// TwinCAT 3 PLC project SPS
// ProgramVersion: 3.1.4023.0
// libraries:
//   Tc2_Standard, * (Beckhoff Automation GmbH)
//   Tc2_System, * (Beckhoff Automation GmbH)
//   Tc2_TcpIp, * (Beckhoff Automation GmbH)
//   Tc2_Utilities, * (Beckhoff Automation GmbH)
//   Tc3_Module, * (Beckhoff Automation GmbH)
// project tree:
//   DUTs/ OBIS_Datatype.TcDUT
//   / PlcTask.TcTTO
//   POUs/ EL3443_OBIS.TcPOU, FB_OBIS.TcPOU, FB_SPEEDWIRE.TcPOU, MAIN.TcPOU, UnixTimestamp.TcPOU
// real-time tasks:
//   TASK PlcTask: cycle T#10ms, priority 20, ADS port 350
// I/O:
//   DEVICE Gerät 1 (EtherCAT), AmsNetId 172.17.204.224.2.1
//     Klemme 1 (EK1100) [EK1100 EtherCAT-Koppler (2A E-Bus)]
//       Klemme 2 (EL3443) [EL3443 3K. Leistungsmessung]
// variable links:
//   SPS/SPS Instance <-> Device 1 (EtherCAT)/Term 1 (EK1100)/Term 2 (EL3443)
//     PlcTask Inputs/MAIN.EL3443_Terminal.MDP5001_341_Input/MDP5001_341_L1_Basic_Current <-> L1 Basic/Current
//     PlcTask Inputs/MAIN.EL3443_Terminal.MDP5001_341_Input/MDP5001_341_L2_Basic_Current <-> L2 Basic/Current
//     PlcTask Inputs/MAIN.EL3443_Terminal.MDP5001_341_Input/MDP5001_341_L3_Basic_Current <-> L3 Basic/Current
//     PlcTask Inputs/MAIN.EL3443_Terminal.MDP5001_341_Input/MDP5001_341_L1_Basic_Voltage <-> L1 Basic/Voltage
//     PlcTask Inputs/MAIN.EL3443_Terminal.MDP5001_341_Input/MDP5001_341_L2_Basic_Voltage <-> L2 Basic/Voltage
//     PlcTask Inputs/MAIN.EL3443_Terminal.MDP5001_341_Input/MDP5001_341_L3_Basic_Voltage <-> L3 Basic/Voltage
//     PlcTask Inputs/MAIN.EL3443_Terminal.MDP5001_341_Input/MDP5001_341_L1_Power_Active_Power <-> L1 Power/Active Power
//     PlcTask Inputs/MAIN.EL3443_Terminal.MDP5001_341_Input/MDP5001_341_L2_Power_Active_Power <-> L2 Power/Active Power
//     PlcTask Inputs/MAIN.EL3443_Terminal.MDP5001_341_Input/MDP5001_341_L3_Power_Active_Power <-> L3 Power/Active Power
//     PlcTask Inputs/MAIN.EL3443_Terminal.MDP5001_341_Input/MDP5001_341_L1_Power_Apparent_Power <-> L1 Power/Apparent Power
//     PlcTask Inputs/MAIN.EL3443_Terminal.MDP5001_341_Input/MDP5001_341_L2_Power_Apparent_Power <-> L2 Power/Apparent Power
//     PlcTask Inputs/MAIN.EL3443_Terminal.MDP5001_341_Input/MDP5001_341_L3_Power_Apparent_Power <-> L3 Power/Apparent Power
//     PlcTask Inputs/MAIN.EL3443_Terminal.MDP5001_341_Input/MDP5001_341_L1_Power_Power_Factor <-> L1 Power/Power Factor
//     PlcTask Inputs/MAIN.EL3443_Terminal.MDP5001_341_Input/MDP5001_341_L2_Power_Power_Factor <-> L2 Power/Power Factor
//     PlcTask Inputs/MAIN.EL3443_Terminal.MDP5001_341_Input/MDP5001_341_L3_Power_Power_Factor <-> L3 Power/Power Factor
//     PlcTask Inputs/MAIN.EL3443_Terminal.MDP5001_341_Input/MDP5001_341_L1_Power_Reactive_Power <-> L1 Power/Reactive Power
//     PlcTask Inputs/MAIN.EL3443_Terminal.MDP5001_341_Input/MDP5001_341_L2_Power_Reactive_Power <-> L2 Power/Reactive Power
//     PlcTask Inputs/MAIN.EL3443_Terminal.MDP5001_341_Input/MDP5001_341_L3_Power_Reactive_Power <-> L3 Power/Reactive Power
//     PlcTask Inputs/MAIN.EL3443_Terminal.MDP5001_341_Input/MDP5001_341_L1_Status_Current_Guard_Error <-> L1 Status/Current Guard Error
//     PlcTask Inputs/MAIN.EL3443_Terminal.MDP5001_341_Input/MDP5001_341_L2_Status_Current_Guard_Error <-> L2 Status/Current Guard Error
//     PlcTask Inputs/MAIN.EL3443_Terminal.MDP5001_341_Input/MDP5001_341_L3_Status_Current_Guard_Error <-> L3 Status/Current Guard Error
//     PlcTask Inputs/MAIN.EL3443_Terminal.MDP5001_341_Input/MDP5001_341_L1_Status_Current_Guard_Warning <-> L1 Status/Current Guard Warning
//     PlcTask Inputs/MAIN.EL3443_Terminal.MDP5001_341_Input/MDP5001_341_L2_Status_Current_Guard_Warning <-> L2 Status/Current Guard Warning
//     PlcTask Inputs/MAIN.EL3443_Terminal.MDP5001_341_Input/MDP5001_341_L3_Status_Current_Guard_Warning <-> L3 Status/Current Guard Warning
//     PlcTask Inputs/MAIN.EL3443_Terminal.MDP5001_341_Input/MDP5001_341_L1_Status_Inaccurate_Current <-> L1 Status/Inaccurate Current
//     PlcTask Inputs/MAIN.EL3443_Terminal.MDP5001_341_Input/MDP5001_341_L2_Status_Inaccurate_Current <-> L2 Status/Inaccurate Current
//     PlcTask Inputs/MAIN.EL3443_Terminal.MDP5001_341_Input/MDP5001_341_L3_Status_Inaccurate_Current <-> L3 Status/Inaccurate Current
//     PlcTask Inputs/MAIN.EL3443_Terminal.MDP5001_341_Input/MDP5001_341_L1_Status_Inaccurate_Voltage <-> L1 Status/Inaccurate Voltage
//     PlcTask Inputs/MAIN.EL3443_Terminal.MDP5001_341_Input/MDP5001_341_L2_Status_Inaccurate_Voltage <-> L2 Status/Inaccurate Voltage
//     PlcTask Inputs/MAIN.EL3443_Terminal.MDP5001_341_Input/MDP5001_341_L3_Status_Inaccurate_Voltage <-> L3 Status/Inaccurate Voltage
//     PlcTask Inputs/MAIN.EL3443_Terminal.MDP5001_341_Input/MDP5001_341_L1_Status_Overcurrent <-> L1 Status/Overcurrent
//     PlcTask Inputs/MAIN.EL3443_Terminal.MDP5001_341_Input/MDP5001_341_L2_Status_Overcurrent <-> L2 Status/Overcurrent
//     PlcTask Inputs/MAIN.EL3443_Terminal.MDP5001_341_Input/MDP5001_341_L3_Status_Overcurrent <-> L3 Status/Overcurrent
//     PlcTask Inputs/MAIN.EL3443_Terminal.MDP5001_341_Input/MDP5001_341_L1_Status_Overvoltage <-> L1 Status/Overvoltage
//     PlcTask Inputs/MAIN.EL3443_Terminal.MDP5001_341_Input/MDP5001_341_L2_Status_Overvoltage <-> L2 Status/Overvoltage
//     PlcTask Inputs/MAIN.EL3443_Terminal.MDP5001_341_Input/MDP5001_341_L3_Status_Overvoltage <-> L3 Status/Overvoltage
//     PlcTask Inputs/MAIN.EL3443_Terminal.MDP5001_341_Input/MDP5001_341_L1_Status_TxPDO_Toggle <-> L1 Status/TxPDO Toggle
//     PlcTask Inputs/MAIN.EL3443_Terminal.MDP5001_341_Input/MDP5001_341_L2_Status_TxPDO_Toggle <-> L2 Status/TxPDO Toggle
//     PlcTask Inputs/MAIN.EL3443_Terminal.MDP5001_341_Input/MDP5001_341_L3_Status_TxPDO_Toggle <-> L3 Status/TxPDO Toggle
//     PlcTask Inputs/MAIN.EL3443_Terminal.MDP5001_341_Input/MDP5001_341_L1_Status_Voltage_Guard_Error <-> L1 Status/Voltage Guard Error
//     PlcTask Inputs/MAIN.EL3443_Terminal.MDP5001_341_Input/MDP5001_341_L2_Status_Voltage_Guard_Error <-> L2 Status/Voltage Guard Error
//     PlcTask Inputs/MAIN.EL3443_Terminal.MDP5001_341_Input/MDP5001_341_L3_Status_Voltage_Guard_Error <-> L3 Status/Voltage Guard Error
//     PlcTask Inputs/MAIN.EL3443_Terminal.MDP5001_341_Input/MDP5001_341_L1_Status_Voltage_Guard_Warning <-> L1 Status/Voltage Guard Warning
//     PlcTask Inputs/MAIN.EL3443_Terminal.MDP5001_341_Input/MDP5001_341_L2_Status_Voltage_Guard_Warning <-> L2 Status/Voltage Guard Warning
//     PlcTask Inputs/MAIN.EL3443_Terminal.MDP5001_341_Input/MDP5001_341_L3_Status_Voltage_Guard_Warning <-> L3 Status/Voltage Guard Warning
//     PlcTask Inputs/MAIN.EL3443_Terminal.MDP5001_341_Input/MDP5001_341_L1_Status_Voltage_Sign_Bit <-> L1 Status/Voltage Sign Bit
//     PlcTask Inputs/MAIN.EL3443_Terminal.MDP5001_341_Input/MDP5001_341_L2_Status_Voltage_Sign_Bit <-> L2 Status/Voltage Sign Bit
//     PlcTask Inputs/MAIN.EL3443_Terminal.MDP5001_341_Input/MDP5001_341_L3_Status_Voltage_Sign_Bit <-> L3 Status/Voltage Sign Bit
//     PlcTask Inputs/MAIN.EL3443_Terminal.MDP5001_341_Input/MDP5001_341_L3_Statistic_Current_Current_Peak <-> L3 Statistic Current/Current Peak
//     PlcTask Inputs/MAIN.EL3443_Terminal.MDP5001_341_Input/MDP5001_341_L3_Statistic_Current_Current_RMS_Maximum <-> L3 Statistic Current/Current RMS Maximum
//     PlcTask Inputs/MAIN.EL3443_Terminal.MDP5001_341_Input/MDP5001_341_L3_Statistic_Current_Current_RMS_Minimum <-> L3 Statistic Current/Current RMS Minimum
//     PlcTask Inputs/MAIN.EL3443_Terminal.MDP5001_341_Input/MDP5001_341_L3_Statistic_Power_Active_Power_Avg <-> L3 Statistic Power/Active Power Avg
//     PlcTask Inputs/MAIN.EL3443_Terminal.MDP5001_341_Input/MDP5001_341_L3_Statistic_Power_Active_Power_Max <-> L3 Statistic Power/Active Power Max
//     PlcTask Inputs/MAIN.EL3443_Terminal.MDP5001_341_Input/MDP5001_341_L3_Statistic_Power_Active_Power_Min <-> L3 Statistic Power/Active Power Min
//     PlcTask Inputs/MAIN.EL3443_Terminal.MDP5001_341_Input/MDP5001_341_L3_Statistic_Power_Apparent_Power_Avg <-> L3 Statistic Power/Apparent Power Avg
//     PlcTask Inputs/MAIN.EL3443_Terminal.MDP5001_341_Input/MDP5001_341_L3_Statistic_Power_Apparent_Power_Max <-> L3 Statistic Power/Apparent Power Max
//     PlcTask Inputs/MAIN.EL3443_Terminal.MDP5001_341_Input/MDP5001_341_L3_Statistic_Power_Apparent_Power_Min <-> L3 Statistic Power/Apparent Power Min
//     PlcTask Inputs/MAIN.EL3443_Terminal.MDP5001_341_Input/MDP5001_341_L3_Statistic_Power_Reactive_Power_Avg <-> L3 Statistic Power/Reactive Power Avg
//     PlcTask Inputs/MAIN.EL3443_Terminal.MDP5001_341_Input/MDP5001_341_L3_Statistic_Power_Reactive_Power_Max <-> L3 Statistic Power/Reactive Power Max
//     PlcTask Inputs/MAIN.EL3443_Terminal.MDP5001_341_Input/MDP5001_341_L3_Statistic_Power_Reactive_Power_Min <-> L3 Statistic Power/Reactive Power Min
//     PlcTask Inputs/MAIN.EL3443_Terminal.MDP5001_341_Input/MDP5001_341_Total_Active_Active_Energy <-> Total Active/Active Energy
//     PlcTask Inputs/MAIN.EL3443_Terminal.MDP5001_341_Input/MDP5001_341_Total_Active_Active_Negative_Energy <-> Total Active/Active Negative Energy
//     PlcTask Inputs/MAIN.EL3443_Terminal.MDP5001_341_Input/MDP5001_341_Total_Active_Active_Positive_Energy <-> Total Active/Active Positive Energy
//     PlcTask Inputs/MAIN.EL3443_Terminal.MDP5001_341_Input/MDP5001_341_Total_Active_Active_Power <-> Total Active/Active Power
//     PlcTask Inputs/MAIN.EL3443_Terminal.MDP5001_341_Input/MDP5001_341_Total_Apparent_Apparent_Energy <-> Total Apparent/Apparent Energy
//     PlcTask Inputs/MAIN.EL3443_Terminal.MDP5001_341_Input/MDP5001_341_Total_Apparent_Apparent_Negative_Energy <-> Total Apparent/Apparent Negative Energy
//     PlcTask Inputs/MAIN.EL3443_Terminal.MDP5001_341_Input/MDP5001_341_Total_Apparent_Apparent_Positive_Energy <-> Total Apparent/Apparent Positive Energy
//     PlcTask Inputs/MAIN.EL3443_Terminal.MDP5001_341_Input/MDP5001_341_Total_Apparent_Apparent_Power <-> Total Apparent/Apparent Power
//     PlcTask Inputs/MAIN.EL3443_Terminal.MDP5001_341_Input/MDP5001_341_Total_Basic_Calculated_Neutral_Line_Current <-> Total Basic/Calculated Neutral Line Current
//     PlcTask Inputs/MAIN.EL3443_Terminal.MDP5001_341_Input/MDP5001_341_Total_Basic_Frequency <-> Total Basic/Frequency
//     PlcTask Inputs/MAIN.EL3443_Terminal.MDP5001_341_Input/MDP5001_341_Total_Basic_Power_Factor <-> Total Basic/Power Factor
//     PlcTask Inputs/MAIN.EL3443_Terminal.MDP5001_341_Input/MDP5001_341_Total_Reactive_Reactive_Energy <-> Total Reactive/Reactive Energy
//     PlcTask Inputs/MAIN.EL3443_Terminal.MDP5001_341_Input/MDP5001_341_Total_Reactive_Reactive_Negative_Energy <-> Total Reactive/Reactive Negative Energy
//     PlcTask Inputs/MAIN.EL3443_Terminal.MDP5001_341_Input/MDP5001_341_Total_Reactive_Reactive_Positive_Energy <-> Total Reactive/Reactive Positive Energy
//     PlcTask Inputs/MAIN.EL3443_Terminal.MDP5001_341_Input/MDP5001_341_Total_Reactive_Reactive_Power <-> Total Reactive/Reactive Power
//     PlcTask Inputs/MAIN.EL3443_Terminal.MDP5001_341_Input/MDP5001_341_Total_Status_Active_Power_Guard_Error <-> Total Status/Active Power Guard Error
//     PlcTask Inputs/MAIN.EL3443_Terminal.MDP5001_341_Input/MDP5001_341_Total_Status_Active_Power_Guard_Warning <-> Total Status/Active Power Guard Warning
//     PlcTask Inputs/MAIN.EL3443_Terminal.MDP5001_341_Input/MDP5001_341_Total_Status_Apparent_Power_Guard_Error <-> Total Status/Apparent Power Guard Error
//     PlcTask Inputs/MAIN.EL3443_Terminal.MDP5001_341_Input/MDP5001_341_Total_Status_Apparent_Power_Guard_Warning <-> Total Status/Apparent Power Guard Warning
//     PlcTask Inputs/MAIN.EL3443_Terminal.MDP5001_341_Input/MDP5001_341_Total_Status_Frequency_Guard_Error <-> Total Status/Frequency Guard Error
//     PlcTask Inputs/MAIN.EL3443_Terminal.MDP5001_341_Input/MDP5001_341_Total_Status_Frequency_Guard_Warning <-> Total Status/Frequency Guard Warning
//     PlcTask Inputs/MAIN.EL3443_Terminal.MDP5001_341_Input/MDP5001_341_Total_Status_Grid_Direction <-> Total Status/Grid Direction
//     PlcTask Inputs/MAIN.EL3443_Terminal.MDP5001_341_Input/MDP5001_341_Total_Status_Neutral_Current_Guard_Error <-> Total Status/Neutral Current Guard Error
//     PlcTask Inputs/MAIN.EL3443_Terminal.MDP5001_341_Input/MDP5001_341_Total_Status_Neutral_Current_Guard_Warning <-> Total Status/Neutral Current Guard Warning
//     PlcTask Inputs/MAIN.EL3443_Terminal.MDP5001_341_Input/MDP5001_341_Total_Status_Power_Quality_Factor <-> Total Status/Power Quality Factor
//     PlcTask Inputs/MAIN.EL3443_Terminal.MDP5001_341_Input/MDP5001_341_Total_Status_Power_Quality_Guard_Error <-> Total Status/Power Quality Guard Error
//     PlcTask Inputs/MAIN.EL3443_Terminal.MDP5001_341_Input/MDP5001_341_Total_Status_Power_Quality_Guard_Warning <-> Total Status/Power Quality Guard Warning
//     PlcTask Inputs/MAIN.EL3443_Terminal.MDP5001_341_Input/MDP5001_341_Total_Status_System_State <-> Total Status/System State
//     PlcTask Inputs/MAIN.EL3443_Terminal.MDP5001_341_Input/MDP5001_341_Total_Status_TxPDO_State <-> Total Status/TxPDO State
//     PlcTask Inputs/MAIN.EL3443_Terminal.MDP5001_341_Input/MDP5001_341_Total_Status_TxPDO_Toggle <-> Total Status/TxPDO Toggle

CONFIGURATION SPS
    RESOURCE PLC ON TwinCAT3
        TASK PlcTask(INTERVAL := T#10ms, PRIORITY := 20);
        PROGRAM MAIN WITH PlcTask : MAIN;
    END_RESOURCE
END_CONFIGURATION

// ---- DUTs/OBIS_Datatype.TcDUT
{attribute 'qualified_only'}
{attribute 'strict'}
TYPE OBIS_Datatype :
(
	TOTAL_ActivePowerPositive := 0,
	TOTAL_ActivePowerNegative := 1,
	TOTAL_ActiveEnergyPositive := 2, 
	TOTAL_ActiveEnergyNegative := 3,
	TOTAL_ApparentPowerPositive := 4,
	TOTAL_ApparentPowerNegative := 5,
	TOTAL_ApparentEnergyPositive := 6, 
	TOTAL_ApparentEnergyNegative := 7,
	TOTAL_ReactivePowerPositive := 8,
	TOTAL_ReactivePowerNegative := 9,
	TOTAL_ReactiveEnergyPositive := 10, 
	TOTAL_ReactiveEnergyNegative := 11,
	TOTAL_PowerFactor := 12,
	TOTAL_Frequency := 13, 
	
	L1_ActivePowerPositive := 14,
	L1_ActivePowerNegative := 15,
	L1_ActiveEnergyPositive := 16, 
	L1_ActiveEnergyNegative := 17,
	L1_ApparentPowerPositive := 18,
	L1_ApparentPowerNegative := 19,
	L1_ApparentEnergyPositive := 20, 
	L1_ApparentEnergyNegative := 21,
	L1_ReactivePowerPositive := 22,
	L1_ReactivePowerNegative := 23,
	L1_ReactiveEnergyPositive := 24, 
	L1_ReactiveEnergyNegative := 25,
	L1_Current := 26,
	L1_Voltage := 27,
	L1_PowerFactor := 28,
	
	L2_ActivePowerPositive := 29,
	L2_ActivePowerNegative := 30,
	L2_ActiveEnergyPositive := 31, 
	L2_ActiveEnergyNegative := 32,
	L2_ApparentPowerPositive := 33,
	L2_ApparentPowerNegative := 34,
	L2_ApparentEnergyPositive := 35, 
	L2_ApparentEnergyNegative := 36,
	L2_ReactivePowerPositive := 37,
	L2_ReactivePowerNegative := 38,
	L2_ReactiveEnergyPositive := 39, 
	L2_ReactiveEnergyNegative := 40,
	L2_Current := 41,
	L2_Voltage := 42,
	L2_PowerFactor := 43,
	
	L3_ActivePowerPositive := 44,
	L3_ActivePowerNegative := 45,
	L3_ActiveEnergyPositive := 46, 
	L3_ActiveEnergyNegative := 47,
	L3_ApparentPowerPositive := 48,
	L3_ApparentPowerNegative := 49,
	L3_ApparentEnergyPositive := 50, 
	L3_ApparentEnergyNegative := 51,
	L3_ReactivePowerPositive := 52,
	L3_ReactivePowerNegative := 53,
	L3_ReactiveEnergyPositive := 54, 
	L3_ReactiveEnergyNegative := 55,
	L3_Current := 56,
	L3_Voltage := 57,
	L3_PowerFactor := 58
	
	
);
END_TYPE

// ---- POUs/MAIN.TcPOU
PROGRAM MAIN
VAR
	//Devices
	EL3443_Terminal			: MDP5001_341_A3044239;
	fbspeedwire				: FB_SPEEDWIRE;
END_VAR

fbspeedwire(
	EL3443 := EL3443_Terminal
	);

END_PROGRAM

// ---- POUs/FB_SPEEDWIRE.TcPOU
FUNCTION_BLOCK FB_SPEEDWIRE
VAR_INPUT
	bEnable					: BOOL 	:= TRUE;
	nLocalPort				: UDINT := 9522;
	sLocalHost				: T_IPv4Addr := '192.168.0.227';(* Adapt local IP address to your device *)
	nRemotePort				: UDINT := 9522;
	sMulticastAddr			: T_IPv4Addr := '239.12.255.254';
	
	EL3443		: MDP5001_341_A3044239;
END_VAR
VAR_OUTPUT
END_VAR
VAR
	fbUdpCreate 			: FB_SocketUdpCreate;
	fbSocketAddMulticast 	: FB_SocketUdpAddMulticastAddress;
	fbSocketDropMulticast 	: FB_SocketUdpDropMulticastAddress;
	fbSocketSend  			: FB_SocketUdpSendTo;
	fbSocketReceive 		: FB_SocketUdpReceiveFrom;
	fbSocketClose			: FB_SocketClose;
	fbCloseAll				: FB_SocketCloseAll;
	bInitialize				: BOOL := TRUE;
	bUdpCreated				: BOOL;
	bMulticastAdded			: BOOL; 
	
	nCounterIn 				: UDINT;
	nCounterOut 			: UDINT;
	nState 					: INT;		
	
	fbEL3443_2_OBIS			: EL3443_OBIS;
	
	send_ton 				: TON;
END_VAR

IF bInitialize = TRUE THEN
(* On PLC reset or program download close all opened/created sockets *)
	fbCloseAll( bExecute:= bInitialize );
	IF fbCloseAll.bBusy OR fbCloseAll.bError THEN
	//	RETURN;
	END_IF
	bInitialize := FALSE;
END_IF






CASE nState OF
0:
	IF bEnable THEN
		bUdpCreated := FALSE;
		bMulticastAdded := FALSE;
		nState := 1;
	END_IF
1:
	fbUdpCreate( bExecute := FALSE );
	fbUdpCreate( nLocalPort := nLocalPort, sLocalHost := sLocalHost, bExecute := TRUE);
	nState := 2;
2:
	fbUdpCreate( bExecute := FALSE );
	IF NOT fbUdpCreate.bBusy THEN
		IF NOT fbUdpCreate.bError THEN
			bUdpCreated := TRUE;
			fbSocketAddMulticast( bExecute := FALSE );
			fbSocketAddMulticast( hSocket := fbUdpCreate.hSocket, sMulticastAddr := sMulticastAddr, bExecute := TRUE );
			nState := 3;
		ELSE
			nState := 100;
		END_IF
	END_IF
3:
	fbSocketAddMulticast( bExecute := FALSE );
	IF NOT fbSocketAddMulticast.bBusy THEN
		IF NOT fbSocketAddMulticast.bError THEN
			bMulticastAdded := TRUE;
			nState := 4;
		ELSE
			nState := 100;
		END_IF
	END_IF
	
4:
	IF bEnable THEN
		nCounterOut := nCounterOut + 1;
		fbSocketSend( bExecute := FALSE );
		fbEL3443_2_OBIS(EL3443 := EL3443);
		fbSocketSend( nRemotePort := nRemotePort, sRemoteHost := sMulticastAddr, hSocket := fbUdpCreate.hSocket, cbLen:= fbEL3443_2_OBIS.GetDataLength(), pSrc := fbEL3443_2_OBIS.GetData(), bExecute := TRUE );
		nState := 5;
	ELSE
		nState := 10;
	END_IF
5:
	fbSocketSend( bExecute := FALSE );
	IF NOT fbSocketSend.bBusy THEN
		IF NOT fbSocketSend.bError THEN
			nState := 6;
		ELSE
 			nState := 100;
		END_IF
	END_IF
6:	
	fbSocketReceive( bExecute := FALSE );
	IF NOT fbSocketReceive.bBusy THEN
		IF NOT fbSocketReceive.bError THEN
			nState:= 7;
			
		ELSE
			nState := 100;
		END_IF
	END_IF

7:	send_ton(IN := TRUE, PT:= T#200MS);
	IF send_ton.Q THEN
		nState:= 4;
		send_ton(IN:=FALSE);
	END_IF
	
10:
	fbSocketDropMulticast( bExecute := FALSE );
	fbSocketDropMulticast( hSocket := fbUdpCreate.hSocket, sMulticastAddr := sMulticastAddr, bExecute := TRUE );
	nState := 11;
11:	
	fbSocketDropMulticast( bExecute := FALSE );
	IF NOT fbSocketDropMulticast.bBusy THEN
		bMulticastAdded := FALSE;
		IF NOT fbSocketDropMulticast.bError THEN
			nState := 20;
		ELSE
			nState := 100;
		END_IF
	END_IF

20:	
	fbSocketClose( bExecute := FALSE );
	fbSocketClose( hSocket := fbUdpCreate.hSocket, bExecute := TRUE );
	nState := 21;
21:	
	fbSocketClose( bExecute := FALSE );
	IF NOT fbSocketClose.bBusy THEN
		bUdpCreated := FALSE;
		IF NOT fbSocketClose.bError THEN
			nState := 0;	
		ELSE
			nState := 100;	
		END_IF
	END_IF
	
100:
	IF bMulticastAdded THEN
		nState := 10;
	ELSIF bUdpCreated THEN
		nState := 20;
	ELSE
		nState := 0;
	END_IF
	
END_CASE

END_FUNCTION_BLOCK

// ---- POUs/EL3443_OBIS.TcPOU
FUNCTION_BLOCK EL3443_OBIS
VAR_INPUT
	EL3443 : MDP5001_341_A3044239;
END_VAR
VAR_OUTPUT
END_VAR
VAR
	unixTime: UnixTimestamp;
    timestampSeconds: ULINT;
    timestampMilliseconds: ULINT;
	
	obis_data : FB_OBIS;	
END_VAR

unixTime();
timestampMilliseconds := unixTime.milliseconds;
timestampSeconds := unixTime.seconds;

obis_data.addTime(u32time := ULINT_TO_UDINT(timestampMilliseconds));

//L1------------------------------------------------

obis_data.Addfloat(datatype := OBIS_Datatype.L1_Voltage, floatdata := EL3443.MDP5001_341_Input.MDP5001_341_L1_Basic_Voltage);
obis_data.Addfloat(datatype := OBIS_Datatype.L1_Current, floatdata := EL3443.MDP5001_341_Input.MDP5001_341_L1_Basic_Current);
obis_data.Addfloat(datatype := OBIS_Datatype.L1_PowerFactor, floatdata := EL3443.MDP5001_341_Input.MDP5001_341_L1_Power_Power_Factor);

IF EL3443.MDP5001_341_Input.MDP5001_341_L1_Power_Active_Power > 0.0 THEN
	obis_data.Addfloat(datatype := OBIS_Datatype.L1_ActivePowerPositive, floatdata := EL3443.MDP5001_341_Input.MDP5001_341_L1_Power_Active_Power);
	obis_data.Addfloat(datatype := OBIS_Datatype.L1_ActivePowerNegative, floatdata := 0.0);
ELSE
	obis_data.Addfloat(datatype := OBIS_Datatype.L1_ActivePowerPositive, floatdata := 0.0);
	obis_data.Addfloat(datatype := OBIS_Datatype.L1_ActivePowerNegative, floatdata := -EL3443.MDP5001_341_Input.MDP5001_341_L1_Power_Active_Power);	
END_IF

IF EL3443.MDP5001_341_Input.MDP5001_341_L1_Power_Apparent_Power > 0.0 THEN
	obis_data.Addfloat(datatype := OBIS_Datatype.L1_ApparentPowerPositive, floatdata := EL3443.MDP5001_341_Input.MDP5001_341_L1_Power_Apparent_Power);
	obis_data.Addfloat(datatype := OBIS_Datatype.L1_ApparentPowerNegative, floatdata := 0.0);
ELSE
	obis_data.Addfloat(datatype := OBIS_Datatype.L1_ApparentPowerPositive, floatdata := 0.0);
	obis_data.Addfloat(datatype := OBIS_Datatype.L1_ApparentPowerNegative, floatdata := -EL3443.MDP5001_341_Input.MDP5001_341_L1_Power_Apparent_Power);	
END_IF

IF EL3443.MDP5001_341_Input.MDP5001_341_L1_Power_Reactive_Power > 0.0 THEN
	obis_data.Addfloat(datatype := OBIS_Datatype.L1_ReactivePowerPositive, floatdata := EL3443.MDP5001_341_Input.MDP5001_341_L1_Power_Reactive_Power);
	obis_data.Addfloat(datatype := OBIS_Datatype.L1_ReactivePowerNegative, floatdata := 0.0);
ELSE
	obis_data.Addfloat(datatype := OBIS_Datatype.L1_ReactivePowerPositive, floatdata := 0.0);
	obis_data.Addfloat(datatype := OBIS_Datatype.L1_ReactivePowerNegative, floatdata := -EL3443.MDP5001_341_Input.MDP5001_341_L1_Power_Reactive_Power);	
END_IF


(*
obis_data.AddUint64(datatype := OBIS_Datatype.L1_ActiveEnergyPositive, u64data := 0);
obis_data.AddUint64(datatype := OBIS_Datatype.L1_ActiveEnergyNegative, u64data := 0);
obis_data.AddUint64(datatype := OBIS_Datatype.L1_ApparentEnergyPositive, u64data := 0);
obis_data.AddUint64(datatype := OBIS_Datatype.L1_ApparentEnergyNegative, u64data := 0);
obis_data.AddUint64(datatype := OBIS_Datatype.L1_ReactiveEnergyPositive, u64data := 0);
obis_data.AddUint64(datatype := OBIS_Datatype.L1_ReactiveEnergyNegative, u64data := 0);

*)

//L2------------------------------------------------

obis_data.Addfloat(datatype := OBIS_Datatype.L2_Voltage, floatdata := EL3443.MDP5001_341_Input.MDP5001_341_L2_Basic_Voltage);
obis_data.Addfloat(datatype := OBIS_Datatype.L2_Current, floatdata := EL3443.MDP5001_341_Input.MDP5001_341_L2_Basic_Current);
obis_data.Addfloat(datatype := OBIS_Datatype.L2_PowerFactor, floatdata := EL3443.MDP5001_341_Input.MDP5001_341_L2_Power_Power_Factor);

IF EL3443.MDP5001_341_Input.MDP5001_341_L2_Power_Active_Power > 0.0 THEN
	obis_data.Addfloat(datatype := OBIS_Datatype.L2_ActivePowerPositive, floatdata := EL3443.MDP5001_341_Input.MDP5001_341_L2_Power_Active_Power);
	obis_data.Addfloat(datatype := OBIS_Datatype.L2_ActivePowerNegative, floatdata := 0.0);
ELSE
	obis_data.Addfloat(datatype := OBIS_Datatype.L2_ActivePowerPositive, floatdata := 0.0);
	obis_data.Addfloat(datatype := OBIS_Datatype.L2_ActivePowerNegative, floatdata := -EL3443.MDP5001_341_Input.MDP5001_341_L2_Power_Active_Power);	
END_IF

IF EL3443.MDP5001_341_Input.MDP5001_341_L2_Power_Apparent_Power > 0.0 THEN
	obis_data.Addfloat(datatype := OBIS_Datatype.L2_ApparentPowerPositive, floatdata := EL3443.MDP5001_341_Input.MDP5001_341_L2_Power_Apparent_Power);
	obis_data.Addfloat(datatype := OBIS_Datatype.L2_ApparentPowerNegative, floatdata := 0.0);
ELSE
	obis_data.Addfloat(datatype := OBIS_Datatype.L2_ApparentPowerPositive, floatdata := 0.0);
	obis_data.Addfloat(datatype := OBIS_Datatype.L2_ApparentPowerNegative, floatdata := -EL3443.MDP5001_341_Input.MDP5001_341_L2_Power_Apparent_Power);	
END_IF

IF EL3443.MDP5001_341_Input.MDP5001_341_L2_Power_Reactive_Power > 0.0 THEN
	obis_data.Addfloat(datatype := OBIS_Datatype.L2_ReactivePowerPositive, floatdata := EL3443.MDP5001_341_Input.MDP5001_341_L2_Power_Reactive_Power);
	obis_data.Addfloat(datatype := OBIS_Datatype.L2_ReactivePowerNegative, floatdata := 0.0);
ELSE
	obis_data.Addfloat(datatype := OBIS_Datatype.L2_ReactivePowerPositive, floatdata := 0.0);
	obis_data.Addfloat(datatype := OBIS_Datatype.L2_ReactivePowerNegative, floatdata := -EL3443.MDP5001_341_Input.MDP5001_341_L2_Power_Reactive_Power);	
END_IF

(*
obis_data.AddUint64(datatype := OBIS_Datatype.L2_ActiveEnergyPositive, u64data := 0);
obis_data.AddUint64(datatype := OBIS_Datatype.L2_ActiveEnergyNegative, u64data := 0);
obis_data.AddUint64(datatype := OBIS_Datatype.L2_ApparentEnergyPositive, u64data := 0);
obis_data.AddUint64(datatype := OBIS_Datatype.L2_ApparentEnergyNegative, u64data := 0);
obis_data.AddUint64(datatype := OBIS_Datatype.L2_ReactiveEnergyPositive, u64data := 0);
obis_data.AddUint64(datatype := OBIS_Datatype.L2_ReactiveEnergyNegative, u64data := 0);
*)

//L3------------------------------------------------

obis_data.Addfloat(datatype := OBIS_Datatype.L3_Voltage, floatdata := EL3443.MDP5001_341_Input.MDP5001_341_L3_Basic_Voltage);
obis_data.Addfloat(datatype := OBIS_Datatype.L3_Current, floatdata := EL3443.MDP5001_341_Input.MDP5001_341_L3_Basic_Current);
obis_data.Addfloat(datatype := OBIS_Datatype.L3_PowerFactor, floatdata := EL3443.MDP5001_341_Input.MDP5001_341_L3_Power_Power_Factor);

IF EL3443.MDP5001_341_Input.MDP5001_341_L3_Power_Active_Power > 0.0 THEN
	obis_data.Addfloat(datatype := OBIS_Datatype.L3_ActivePowerPositive, floatdata := EL3443.MDP5001_341_Input.MDP5001_341_L3_Power_Active_Power);
	obis_data.Addfloat(datatype := OBIS_Datatype.L3_ActivePowerNegative, floatdata := 0.0);
ELSE
	obis_data.Addfloat(datatype := OBIS_Datatype.L3_ActivePowerPositive, floatdata := 0.0);
	obis_data.Addfloat(datatype := OBIS_Datatype.L3_ActivePowerNegative, floatdata := -EL3443.MDP5001_341_Input.MDP5001_341_L3_Power_Active_Power);	
END_IF

IF EL3443.MDP5001_341_Input.MDP5001_341_L3_Power_Apparent_Power > 0.0 THEN
	obis_data.Addfloat(datatype := OBIS_Datatype.L3_ApparentPowerPositive, floatdata := EL3443.MDP5001_341_Input.MDP5001_341_L3_Power_Apparent_Power);
	obis_data.Addfloat(datatype := OBIS_Datatype.L3_ApparentPowerNegative, floatdata := 0.0);
ELSE
	obis_data.Addfloat(datatype := OBIS_Datatype.L3_ApparentPowerPositive, floatdata := 0.0);
	obis_data.Addfloat(datatype := OBIS_Datatype.L3_ApparentPowerNegative, floatdata := -EL3443.MDP5001_341_Input.MDP5001_341_L3_Power_Apparent_Power);	
END_IF

IF EL3443.MDP5001_341_Input.MDP5001_341_L3_Power_Reactive_Power > 0.0 THEN
	obis_data.Addfloat(datatype := OBIS_Datatype.L3_ReactivePowerPositive, floatdata := EL3443.MDP5001_341_Input.MDP5001_341_L3_Power_Reactive_Power);
	obis_data.Addfloat(datatype := OBIS_Datatype.L3_ReactivePowerNegative, floatdata := 0.0);
ELSE
	obis_data.Addfloat(datatype := OBIS_Datatype.L3_ReactivePowerPositive, floatdata := 0.0);
	obis_data.Addfloat(datatype := OBIS_Datatype.L3_ReactivePowerNegative, floatdata := -EL3443.MDP5001_341_Input.MDP5001_341_L3_Power_Reactive_Power);	
END_IF

(*
obis_data.AddUint64(datatype := OBIS_Datatype.L3_ActiveEnergyPositive, u64data := 0);
obis_data.AddUint64(datatype := OBIS_Datatype.L3_ActiveEnergyNegative, u64data := 0);
obis_data.AddUint64(datatype := OBIS_Datatype.L3_ApparentEnergyPositive, u64data := 0);
obis_data.AddUint64(datatype := OBIS_Datatype.L3_ApparentEnergyNegative, u64data := 0);
obis_data.AddUint64(datatype := OBIS_Datatype.L3_ReactiveEnergyPositive, u64data := 0);
obis_data.AddUint64(datatype := OBIS_Datatype.L3_ReactiveEnergyNegative, u64data := 0);
*)

//Total------------------------------------------------


obis_data.Addfloat(datatype := OBIS_Datatype.TOTAL_PowerFactor, floatdata := EL3443.MDP5001_341_Input.MDP5001_341_Total_Basic_Power_Factor);
obis_data.Addfloat(datatype := OBIS_Datatype.TOTAL_Frequency, floatdata := EL3443.MDP5001_341_Input.MDP5001_341_Total_Basic_Frequency);

(*
obis_data.AddUint64(datatype := OBIS_Datatype.TOTAL_ActiveEnergyPositive, u64data := EL3443.MDP5001_341_Input.MDP5001_341_Total_Active_Active_Positive_Energy);
obis_data.AddUint64(datatype := OBIS_Datatype.TOTAL_ActiveEnergyNegative, u64data := EL3443.MDP5001_341_Input.MDP5001_341_Total_Active_Active_Negative_Energy);
obis_data.AddUint64(datatype := OBIS_Datatype.TOTAL_ApparentEnergyPositive, u64data := EL3443.MDP5001_341_Input.MDP5001_341_Total_Apparent_Apparent_Positive_Energy);
obis_data.AddUint64(datatype := OBIS_Datatype.TOTAL_ApparentEnergyNegative, u64data := EL3443.MDP5001_341_Input.MDP5001_341_Total_Apparent_Apparent_Negative_Energy);
obis_data.AddUint64(datatype := OBIS_Datatype.TOTAL_ReactiveEnergyPositive, u64data := EL3443.MDP5001_341_Input.MDP5001_341_Total_Reactive_Reactive_Positive_Energy);
obis_data.AddUint64(datatype := OBIS_Datatype.TOTAL_ReactiveEnergyNegative, u64data := EL3443.MDP5001_341_Input.MDP5001_341_Total_Reactive_Reactive_Negative_Energy);
*)

IF EL3443.MDP5001_341_Input.MDP5001_341_Total_Active_Active_Power > 0.0 THEN
	obis_data.Addfloat(datatype := OBIS_Datatype.TOTAL_ActivePowerPositive, floatdata := EL3443.MDP5001_341_Input.MDP5001_341_Total_Active_Active_Power);
	obis_data.Addfloat(datatype := OBIS_Datatype.TOTAL_ActivePowerNegative, floatdata := 0.0);
ELSE
	obis_data.Addfloat(datatype := OBIS_Datatype.TOTAL_ActivePowerPositive, floatdata := 0.0);
	obis_data.Addfloat(datatype := OBIS_Datatype.TOTAL_ActivePowerNegative, floatdata := -EL3443.MDP5001_341_Input.MDP5001_341_Total_Active_Active_Power);	
END_IF

IF EL3443.MDP5001_341_Input.MDP5001_341_Total_Apparent_Apparent_Power > 0.0 THEN
	obis_data.Addfloat(datatype := OBIS_Datatype.TOTAL_ApparentPowerPositive, floatdata := EL3443.MDP5001_341_Input.MDP5001_341_Total_Apparent_Apparent_Power);
	obis_data.Addfloat(datatype := OBIS_Datatype.TOTAL_ApparentPowerNegative, floatdata := 0.0);
ELSE
	obis_data.Addfloat(datatype := OBIS_Datatype.TOTAL_ApparentPowerPositive, floatdata := 0.0);
	obis_data.Addfloat(datatype := OBIS_Datatype.TOTAL_ApparentPowerNegative, floatdata := -EL3443.MDP5001_341_Input.MDP5001_341_Total_Apparent_Apparent_Power);	
END_IF

IF EL3443.MDP5001_341_Input.MDP5001_341_Total_Reactive_Reactive_Power > 0.0 THEN
	obis_data.Addfloat(datatype := OBIS_Datatype.TOTAL_ReactivePowerPositive, floatdata := EL3443.MDP5001_341_Input.MDP5001_341_Total_Reactive_Reactive_Power);
	obis_data.Addfloat(datatype := OBIS_Datatype.TOTAL_ReactivePowerNegative, floatdata := 0.0);
ELSE
	obis_data.Addfloat(datatype := OBIS_Datatype.TOTAL_ReactivePowerPositive, floatdata := 0.0);
	obis_data.Addfloat(datatype := OBIS_Datatype.TOTAL_ReactivePowerNegative, floatdata := -EL3443.MDP5001_341_Input.MDP5001_341_Total_Reactive_Reactive_Power);	
END_IF

METHOD GetData : POINTER TO BYTE
VAR_INPUT
END_VAR
GetData := obis_data.GetData();
END_METHOD

METHOD GetDataLength : UDINT
VAR_INPUT
END_VAR
GetDataLength := 608;
END_METHOD

END_FUNCTION_BLOCK

// ---- POUs/UnixTimestamp.TcPOU
FUNCTION_BLOCK UnixTimestamp
VAR_INPUT
END_VAR
VAR_OUTPUT
	seconds: ULINT;
    milliseconds: ULINT;
END_VAR
VAR
	localSystemTime : FB_LocalSystemTime := ( bEnable := TRUE, dwCycle := 1 );
    getTimeZoneInformation : FB_GetTimeZoneInformation;
    timeZoneInformation : ST_TimeZoneInformation;
    specificLocalTimeToFileTime : FB_TzSpecificLocalTimeToFileTime;
    fileTime: T_FILETIME;
    onZerothSecondLastCycle : BOOL;
END_VAR

// Get local system time
localSystemTime();

// On the zeroth second of each minutesync timezone information
IF (timeZoneInformation.standardName = '' OR (localSystemTime.systemTime.wSecond = 0 AND NOT onZerothSecondLastCycle)) THEN
    getTimeZoneInformation(sNetID := '', bExecute := TRUE, tzInfo => timeZoneInformation);
END_IF;

// Convert local system time to unix timestamps
specificLocalTimeToFileTime(in := Tc2_Utilities.SYSTEMTIME_TO_FILETIME(localSystemTime.systemTime), tzInfo := timeZoneInformation, out => fileTime);
seconds := (SHL(DWORD_TO_ULINT(fileTime.dwHighDateTime), 32) + DWORD_TO_ULINT(fileTime.dwLowDateTime)) / 10000000 - 11644473600;
milliseconds := (SHL(DWORD_TO_ULINT(fileTime.dwHighDateTime), 32) + DWORD_TO_ULINT(fileTime.dwLowDateTime)) / 10000 - 11644473600000;

onZerothSecondLastCycle := localSystemTime.systemTime.wSecond = 0;

END_FUNCTION_BLOCK

// ---- POUs/FB_OBIS.TcPOU
FUNCTION_BLOCK FB_OBIS
VAR_INPUT
END_VAR
VAR_OUTPUT
END_VAR
VAR
	data : ARRAY [0..607] OF BYTE := [83, 77, 65, 0, 0, 4, 2, 160, 0, 0, 0, 1, 2, 76, 0, 16, 96, 105, 1, 93, 113, 87, 157, 42, 145, 195, 170, 229, 0, 1, 4, 0, 0, 0, 4, 192, 0, 1, 8, 0, 0, 0, 0, 1, 27, 80, 113, 64, 0, 2, 4, 0, 0, 0, 0, 0, 0, 2, 8, 0, 0, 0, 0, 0, 65, 115, 204, 96, 0, 3, 4, 0, 0, 0, 0, 0, 0, 3, 8, 0, 0, 0, 0, 0, 1, 68, 24, 192, 0, 4, 4, 0, 0, 0, 7, 97, 0, 4, 8, 0, 0, 0, 0, 0, 203, 199, 123, 0, 0, 9, 4, 0, 0, 0, 8, 198, 0, 9, 8, 0, 0, 0, 0, 1, 121, 25, 106, 32, 0, 10, 4, 0, 0, 0, 0, 0, 0, 10, 8, 0, 0, 0, 0, 0, 70, 76, 180, 64, 0, 13, 4, 0, 0, 0, 2, 28, 0, 14, 4, 0, 0, 0, 195, 240, 0, 21, 4, 0, 0, 0, 0, 0, 0, 21, 8, 0, 0, 0, 0, 0, 72, 109, 19, 160, 0, 22, 4, 0, 0, 0, 0, 217, 0, 22, 8, 0, 0, 0, 0, 0, 30, 95, 6, 64, 0, 23, 4, 0, 0, 0, 0, 0, 0, 23, 8, 0, 0, 0, 0, 0, 0, 136, 59, 0, 0, 24, 4, 0, 0, 0, 0, 223, 0, 24, 8, 0, 0, 0, 0, 0, 37, 222, 86, 0, 0, 29, 4, 0, 0, 0, 0, 0, 0, 29, 8, 0, 0, 0, 0, 0, 101, 164, 5, 0, 0, 30, 4, 0, 0, 0, 1, 55, 0, 30, 8, 0, 0, 0, 0, 0, 30, 244, 112, 63, 0, 31, 4, 0, 0, 0, 0, 180, 0, 32, 4, 0, 0, 3, 138, 34, 0, 33, 4, 0, 0, 0, 2, 188, 0, 41, 4, 0, 0, 0, 6, 72, 0, 41, 8, 0, 0, 0, 0, 0, 166, 88, 167, 224, 0, 42, 4, 0, 0, 0, 0, 0, 0, 42, 8, 0, 0, 0, 0, 0, 16, 177, 174, 128, 0, 43, 4, 0, 0, 0, 0, 0, 0, 43, 8, 0, 0, 0, 0, 0, 1, 149, 101, 64, 0, 44, 4, 0, 0, 0, 4, 236, 0, 44, 8, 0, 0, 0, 0, 0, 114, 214, 221, 96, 0, 49, 4, 0, 0, 0, 7, 251, 0, 49, 8, 0, 0, 0, 0, 0, 209, 9, 218, 224, 0, 50, 4, 0, 0, 0, 0, 0, 0, 50, 8, 0, 0, 0, 0, 0, 19, 30, 104, 192, 0, 51, 4, 0, 0, 0, 4, 96, 0, 52, 4, 0, 0, 3, 133, 4, 0, 53, 4, 0, 0, 0, 3, 22, 0, 61, 4, 0, 0, 0, 0, 0, 0, 61, 8, 0, 0, 0, 0, 0, 58, 50, 2, 159, 0, 62, 4, 0, 0, 0, 0, 176, 0, 62, 8, 0, 0, 0, 0, 0, 32, 9, 215, 224, 0, 63, 4, 0, 0, 0, 0, 0, 0, 63, 8, 0, 0, 0, 0, 0, 0, 93, 98, 64, 0, 64, 4, 0, 0, 0, 1, 150, 0, 64, 8, 0, 0, 0, 0, 0, 52, 73, 49, 96, 0, 69, 4, 0, 0, 0, 0, 0, 0, 69, 8, 0, 0, 0, 0, 0, 93, 66, 99, 192, 0, 70, 4, 0, 0, 0, 1, 187, 0, 70, 8, 0, 0, 0, 0, 0, 33, 166, 237, 224, 0, 71, 4, 0, 0, 0, 0, 230, 0, 72, 4, 0, 0, 3, 130, 202, 0, 73, 4, 0, 0, 0, 1, 144, 144, 0, 0, 0, 2, 0, 18, 82, 0, 0, 0, 0];
	u32tmp : UDINT;
END_VAR


//sma signature
//data[0..3] = 83, 77, 65, 0, 

//sma tag0
//data[4..7] = 0, 4, 2, 160,

//sma group
//data[8..11] = 0, 0, 0, 1, 

//sma length offset
//data[12..13] =  2, 76,

//sma netver
//data[14..15] =  0, 16,

//sma protocol 
//data[16..17] = 96, 105

///Speedwire protocol
//SusyID
//data[18..19] = 1, 93

//SerialNumber
//data[20..23] = 113, 87, 157, 42, 

//Time
//data[24..27] = 145, 195, 170, 229,

//Total active power positive (8byte)
//data[28..35] = 0, 1, 4, 0, 0, 0, 4, 192,

//Total active enregy positive (12 byte)
//data[36..47] =  0, 1, 8, 0, 0, 0, 0, 1, 27, 80, 113, 64,

//Total active power negative (8byte)
//data[48..55] =  0, 2, 4, 0, 0, 0, 0, 0, 

//Total active enregy negative (12 byte)
//data[56..67] = 0,2, 8, 0, 0, 0, 0, 0, 65, 115, 204, 96,

//Total reactive power positive (8 byte)
// data[68..75] = 0, 3, 4, 0, 0, 0, 0, 0,

//Total reactive enegry pisitve (12 byte)
// data[76..87] = 0, 3, 8, 0, 0, 0, 0, 0, 1, 68, 24, 192,

//Total reactive power negative (8 byte)
// data [88..95] = 0, 4, 4, 0, 0, 0, 7, 97,

//Total reactive energy negative (12 byte)
// data[96..107] = 0, 4, 8, 0, 0, 0, 0, 0, 203, 199, 123, 0,

//Total apparent power positive (8byte)
// data[108..115] = 0, 9, 4, 0, 0, 0, 8, 198,

//TOtal apparent energy positiuve (12 byte)
// data[116..127] = 0, 9, 8, 0, 0, 0, 0, 1, 121, 25, 106, 32,

//Total apparent power negative (8 byte)
// data[128..135] = 0, 10, 4, 0, 0, 0, 0, 0, 0,

//Total apparent enegry negative (12 byte)
// data[136..147] = 10, 8, 0, 0, 0, 0, 0, 70, 76, 180, 64,

//Total Power Factor (8 byte)
// data[148..155] = 0, 13, 4, 0, 0, 0, 2, 28,

//Total Frequency
// data[156..163] = 0, 14, 4, 0, 0, 0, 195, 240





//L1 active power positive (8byte)
//data[164..171] = 0, 21, 4, 0, 0, 0, 0, 0,

//L1 active enregy positive (12 byte)
//data[172..183] =  0, 21, 8, 0, 0, 0, 0, 0, 72, 109, 19, 160,

//L1 active power negative (8byte)
//data[184..191] =   0, 22, 4, 0, 0, 0, 0, 217, 

//L1 active enregy negative (12 byte)
//data[192..203] = 0, 22, 8, 0, 0, 0, 0, 0, 30, 95, 6, 64,

//L1 reactive power positive (8 byte)
// data[204..211] = 0, 23, 4, 0, 0, 0, 0, 0,

//L1 reactive enegry pisitve (12 byte)
// data[..87] =  0, 23, 8, 0, 0, 0, 0, 0, 0, 136, 59, 0,

//L1 reactive power negative (8 byte)
// data [..95] =  0, 24, 4, 0, 0, 0, 0, 223,

//L1 reactive energy negative (12 byte)
// data[..107] = 0, 24, 8, 0, 0, 0, 0, 0, 37, 222, 86, 0,

//L1 apparent power positive (8byte)
// data[..115] = 0, 29, 4, 0, 0, 0, 0, 0,

//L1 apparent energy positiuve (12 byte)
// data[..127] = 0, 29, 8, 0, 0, 0, 0, 0, 101, 164, 5, 0,

//L1 apparent power negative (8 byte)
// data[..135] = 0, 30, 4, 0, 0, 0, 1, 55,

//L1 apparent enegry negative (12 byte)
// data[..147] = 0, 30, 8, 0, 0, 0, 0, 0, 30, 244, 112, 63,

//L1 Current
// data[..163] =  0, 31, 4, 0, 0, 0, 0, 180,

//L1 Voltage
// data[..163] = 0, 32, 4, 0, 0, 3, 138, 34, 

//L1 Power Factor (8 byte)
// data[..155] = 0, 33, 4, 0, 0, 0, 2, 188,


//L2 active power positive (8byte)
//data[..35] =  0, 41, 4, 0, 0, 0, 6, 72,

//L2 active enregy positive (12 byte)
//data[..47] = 0, 41, 8, 0, 0, 0, 0, 0, 166, 88, 167, 224,

//L2 active power negative (8byte)
//data[..55] = 0, 42, 4, 0, 0, 0, 0, 0,

//L2 active enregy negative (12 byte)
//data[..67] = 0, 42, 8, 0, 0, 0, 0, 0, 16, 177, 174, 128,

//L2 reactive power positive (8 byte)
// data[..75] =   0, 43, 4, 0, 0, 0, 0, 0,

//L2 reactive enegry pisitve (12 byte)
// data[..87] =  0, 43, 8, 0, 0, 0, 0, 0, 1, 149, 101, 64,

//L2 reactive power negative (8 byte)
// data [..95] = 0, 44, 4, 0, 0, 0, 4, 236,

//L2 reactive energy negative (12 byte)
// data[..107] = 0, 44, 8, 0, 0, 0, 0, 0, 114, 214, 221, 96,

//L2 apparent power positive (8byte)
// data[..115] =  0, 49, 4, 0, 0, 0, 7, 251,

//L2 apparent energy positiuve (12 byte)
// data[..127] =  0, 49, 8, 0, 0, 0, 0, 0, 209, 9, 218, 224,

//L2 apparent power negative (8 byte)
// data[..135] =    0, 50, 4, 0, 0, 0, 0, 0,

//L2 apparent enegry negative (12 byte)
// data[..147] = 0, 50, 8, 0, 0, 0, 0, 0, 19, 30, 104, 192,

//L2 Current
// data[..163] = 0, 51, 4, 0, 0, 0, 4, 96,

//L2 Voltage
// data[..163] = 0, 52, 4, 0, 0, 3, 133, 4,

//L2 Power Factor (8 byte)
// data[..155] =  0, 53, 4, 0, 0, 0, 3, 22,






//L3 active power positive (8byte)
//data[..35] = 0, 61, 4, 0, 0, 0, 0, 0,

//L3 active enregy positive (12 byte)
//data[..47] =   0, 61, 8, 0, 0, 0, 0, 0, 58, 50, 2, 159,

//L3 active power negative (8byte)
//data[..55] =  0, 62, 4, 0, 0, 0, 0, 176,

//L3 active enregy negative (12 byte)
//data[..67] =  0, 62, 8, 0, 0, 0, 0, 0, 32, 9, 215, 224,

//L3 reactive power positive (8 byte)
// data[..75] = 0, 63, 4, 0, 0, 0, 0, 0,

//L3 reactive enegry pisitve (12 byte)
// data[..87] = 0, 63, 8, 0, 0, 0, 0, 0, 0, 93, 98, 64,

//L3 reactive power negative (8 byte)
// data [..95] = 0, 64, 4, 0, 0, 0, 1, 150,

//L3 reactive energy negative (12 byte)
// data[..107] = 0, 64, 8, 0, 0, 0, 0, 0, 52, 73, 49, 96,

//L3 apparent power positive (8byte)
// data[..115] = 0, 69, 4, 0, 0, 0, 0, 0,

//L3 apparent energy positiuve (12 byte)
// data[..127] = 0, 69, 8, 0, 0, 0, 0, 0, 93, 66, 99, 192,

//L3 apparent power negative (8 byte)
// data[..135] =  0, 70, 4, 0, 0, 0, 1, 187,

//L3 apparent enegry negative (12 byte)
// data[..147] = 0, 70, 8, 0, 0, 0, 0, 0, 33, 166, 237, 224,

//L3 Current
// data[..163] = 0, 71, 4, 0, 0, 0, 0, 230,

//L3 Voltage
// data[..163] = 0, 72, 4, 0, 0, 3, 130, 202,

//L3 Power Factor (8 byte)
// data[..155] = 0, 73, 4, 0, 0, 0, 1, 144,


//Firmware Version
//data[] 144, 0, 0, 0, 2, 0, 18, 82,


//End of data
//data = 0, 0, 0, 0

METHOD AddFloat : BOOL
VAR_INPUT
	datatype : OBIS_Datatype;
	floatdata : REAL;	
END_VAR
CASE datatype OF
	OBIS_Datatype.TOTAL_ActivePowerPositive:
		u32tmp := REAL_TO_DWORD(floatdata * 10.0);
		u32tmp := HOST_TO_BE32(in := u32tmp);
		memcpy(srcAddr := ADR(u32tmp), destAddr := ADR(data[32]), n:= 4);

	OBIS_Datatype.TOTAL_ActivePowerNegative:
		u32tmp := REAL_TO_DWORD(floatdata * 10.0);
		u32tmp := HOST_TO_BE32(in := u32tmp);
		memcpy(srcAddr := ADR(u32tmp), destAddr := ADR(data[52]), n:= 4);	
		
	OBIS_Datatype.TOTAL_ReactivePowerPositive:
		u32tmp := REAL_TO_DWORD(floatdata * 10.0);
		u32tmp := HOST_TO_BE32(in := u32tmp);
		memcpy(srcAddr := ADR(u32tmp), destAddr := ADR(data[72]), n:= 4);
	
	OBIS_Datatype.TOTAL_ReactivePowerNegative:
		u32tmp := REAL_TO_DWORD(floatdata * 10.0);
		u32tmp := HOST_TO_BE32(in := u32tmp);
		memcpy(srcAddr := ADR(u32tmp), destAddr := ADR(data[92]), n:= 4);	
		
	OBIS_Datatype.TOTAL_ApparentPowerPositive:
		u32tmp := REAL_TO_DWORD(floatdata * 10.0);
		u32tmp := HOST_TO_BE32(in := u32tmp);
		memcpy(srcAddr := ADR(u32tmp), destAddr := ADR(data[112]), n:= 4);
	
	OBIS_Datatype.TOTAL_ApparentPowerNegative:
		u32tmp := REAL_TO_DWORD(floatdata * 10.0);
		u32tmp := HOST_TO_BE32(in := u32tmp);
		memcpy(srcAddr := ADR(u32tmp), destAddr := ADR(data[132]), n:= 4);	
		
	OBIS_Datatype.TOTAL_PowerFactor:
		u32tmp := REAL_TO_DWORD(floatdata * 1000.0);
		u32tmp := HOST_TO_BE32(in := u32tmp);
		memcpy(srcAddr := ADR(u32tmp), destAddr := ADR(data[152]), n:= 4);	
		
	OBIS_Datatype.TOTAL_Frequency:
		u32tmp := REAL_TO_DWORD(floatdata * 1000.0);
		u32tmp := HOST_TO_BE32(in := u32tmp);
		memcpy(srcAddr := ADR(u32tmp), destAddr := ADR(data[160]), n:= 4);	
		
		
		
	OBIS_Datatype.L1_ActivePowerPositive:
		u32tmp := REAL_TO_DWORD(floatdata * 10.0);
		u32tmp := HOST_TO_BE32(in := u32tmp);
		memcpy(srcAddr := ADR(u32tmp), destAddr := ADR(data[168]), n:= 4);

	OBIS_Datatype.L1_ActivePowerNegative:
		u32tmp := REAL_TO_DWORD(floatdata * 10.0);
		u32tmp := HOST_TO_BE32(in := u32tmp);
		memcpy(srcAddr := ADR(u32tmp), destAddr := ADR(data[188]), n:= 4);	
		
	OBIS_Datatype.L1_ReactivePowerPositive:
		u32tmp := REAL_TO_DWORD(floatdata * 10.0);
		u32tmp := HOST_TO_BE32(in := u32tmp);
		memcpy(srcAddr := ADR(u32tmp), destAddr := ADR(data[208]), n:= 4);
	
	OBIS_Datatype.L1_ReactivePowerNegative:
		u32tmp := REAL_TO_DWORD(floatdata * 10.0);
		u32tmp := HOST_TO_BE32(in := u32tmp);
		memcpy(srcAddr := ADR(u32tmp), destAddr := ADR(data[228]), n:= 4);	
		
	OBIS_Datatype.L1_ApparentPowerPositive:
		u32tmp := REAL_TO_DWORD(floatdata * 10.0);
		u32tmp := HOST_TO_BE32(in := u32tmp);
		memcpy(srcAddr := ADR(u32tmp), destAddr := ADR(data[248]), n:= 4);
	
	OBIS_Datatype.L1_ApparentPowerNegative:
		u32tmp := REAL_TO_DWORD(floatdata * 10.0);
		u32tmp := HOST_TO_BE32(in := u32tmp);
		memcpy(srcAddr := ADR(u32tmp), destAddr := ADR(data[268]), n:= 4);	
		
	OBIS_Datatype.L1_Current:
		u32tmp := REAL_TO_DWORD(floatdata * 1000.0);
		u32tmp := HOST_TO_BE32(in := u32tmp);
		memcpy(srcAddr := ADR(u32tmp), destAddr := ADR(data[288]), n:= 4);	

	OBIS_Datatype.L1_Voltage:
		u32tmp := REAL_TO_DWORD(floatdata * 1000.0);
		u32tmp := HOST_TO_BE32(in := u32tmp);
		memcpy(srcAddr := ADR(u32tmp), destAddr := ADR(data[296]), n:= 4);	

	OBIS_Datatype.L1_PowerFactor:
		u32tmp := REAL_TO_DWORD(floatdata * 1000.0);
		u32tmp := HOST_TO_BE32(in := u32tmp);
		memcpy(srcAddr := ADR(u32tmp), destAddr := ADR(data[304]), n:= 4);		

//--------------------------

	OBIS_Datatype.L2_ActivePowerPositive:
		u32tmp := REAL_TO_DWORD(floatdata * 10.0);
		u32tmp := HOST_TO_BE32(in := u32tmp);
		memcpy(srcAddr := ADR(u32tmp), destAddr := ADR(data[312]), n:= 4);

	OBIS_Datatype.L2_ActivePowerNegative:
		u32tmp := REAL_TO_DWORD(floatdata * 10.0);
		u32tmp := HOST_TO_BE32(in := u32tmp);
		memcpy(srcAddr := ADR(u32tmp), destAddr := ADR(data[332]), n:= 4);	
		
	OBIS_Datatype.L2_ReactivePowerPositive:
		u32tmp := REAL_TO_DWORD(floatdata * 10.0);
		u32tmp := HOST_TO_BE32(in := u32tmp);
		memcpy(srcAddr := ADR(u32tmp), destAddr := ADR(data[352]), n:= 4);
	
	OBIS_Datatype.L2_ReactivePowerNegative:
		u32tmp := REAL_TO_DWORD(floatdata * 10.0);
		u32tmp := HOST_TO_BE32(in := u32tmp);
		memcpy(srcAddr := ADR(u32tmp), destAddr := ADR(data[372]), n:= 4);	
		
	OBIS_Datatype.L2_ApparentPowerPositive:
		u32tmp := REAL_TO_DWORD(floatdata * 10.0);
		u32tmp := HOST_TO_BE32(in := u32tmp);
		memcpy(srcAddr := ADR(u32tmp), destAddr := ADR(data[392]), n:= 4);
	
	OBIS_Datatype.L2_ApparentPowerNegative:
		u32tmp := REAL_TO_DWORD(floatdata * 10.0);
		u32tmp := HOST_TO_BE32(in := u32tmp);
		memcpy(srcAddr := ADR(u32tmp), destAddr := ADR(data[412]), n:= 4);	
		
	OBIS_Datatype.L2_Current:
		u32tmp := REAL_TO_DWORD(floatdata * 1000.0);
		u32tmp := HOST_TO_BE32(in := u32tmp);
		memcpy(srcAddr := ADR(u32tmp), destAddr := ADR(data[432]), n:= 4);	

	OBIS_Datatype.L2_Voltage:
		u32tmp := REAL_TO_DWORD(floatdata * 1000.0);
		u32tmp := HOST_TO_BE32(in := u32tmp);
		memcpy(srcAddr := ADR(u32tmp), destAddr := ADR(data[440]), n:= 4);	

	OBIS_Datatype.L2_PowerFactor:
		u32tmp := REAL_TO_DWORD(floatdata * 1000.0);
		u32tmp := HOST_TO_BE32(in := u32tmp);
		memcpy(srcAddr := ADR(u32tmp), destAddr := ADR(data[448]), n:= 4);	

		

	OBIS_Datatype.L3_ActivePowerPositive:
		u32tmp := REAL_TO_DWORD(floatdata * 10.0);
		u32tmp := HOST_TO_BE32(in := u32tmp);
		memcpy(srcAddr := ADR(u32tmp), destAddr := ADR(data[456]), n:= 4);

	OBIS_Datatype.L3_ActivePowerNegative:
		u32tmp := REAL_TO_DWORD(floatdata * 10.0);
		u32tmp := HOST_TO_BE32(in := u32tmp);
		memcpy(srcAddr := ADR(u32tmp), destAddr := ADR(data[476]), n:= 4);	
		
	OBIS_Datatype.L3_ReactivePowerPositive:
		u32tmp := REAL_TO_DWORD(floatdata * 10.0);
		u32tmp := HOST_TO_BE32(in := u32tmp);
		memcpy(srcAddr := ADR(u32tmp), destAddr := ADR(data[496]), n:= 4);
	
	OBIS_Datatype.L3_ReactivePowerNegative:
		u32tmp := REAL_TO_DWORD(floatdata * 10.0);
		u32tmp := HOST_TO_BE32(in := u32tmp);
		memcpy(srcAddr := ADR(u32tmp), destAddr := ADR(data[516]), n:= 4);	
		
	OBIS_Datatype.L3_ApparentPowerPositive:
		u32tmp := REAL_TO_DWORD(floatdata * 10.0);
		u32tmp := HOST_TO_BE32(in := u32tmp);
		memcpy(srcAddr := ADR(u32tmp), destAddr := ADR(data[536]), n:= 4);
	
	OBIS_Datatype.L3_ApparentPowerNegative:
		u32tmp := REAL_TO_DWORD(floatdata * 10.0);
		u32tmp := HOST_TO_BE32(in := u32tmp);
		memcpy(srcAddr := ADR(u32tmp), destAddr := ADR(data[556]), n:= 4);	
		
	OBIS_Datatype.L3_Current:
		u32tmp := REAL_TO_DWORD(floatdata * 1000.0);
		u32tmp := HOST_TO_BE32(in := u32tmp);
		memcpy(srcAddr := ADR(u32tmp), destAddr := ADR(data[576]), n:= 4);	

	OBIS_Datatype.L3_Voltage:
		u32tmp := REAL_TO_DWORD(floatdata * 1000.0);
		u32tmp := HOST_TO_BE32(in := u32tmp);
		memcpy(srcAddr := ADR(u32tmp), destAddr := ADR(data[582]), n:= 4);	

	OBIS_Datatype.L3_PowerFactor:
		u32tmp := REAL_TO_DWORD(floatdata * 1000.0);
		u32tmp := HOST_TO_BE32(in := u32tmp);
		memcpy(srcAddr := ADR(u32tmp), destAddr := ADR(data[590]), n:= 4);		
END_CASE
END_METHOD

METHOD AddTime : BOOL
VAR_INPUT
	u32time : UDINT;
END_VAR
//Time
//data[24..27] = 145, 195, 170, 229,

u32tmp := HOST_TO_BE32(in := u32time);
memcpy(srcAddr := ADR(u32tmp), destAddr := ADR(data[24]), n:= 4);
END_METHOD

METHOD AddUint64 : BOOL
VAR_INPUT
	datatype : OBIS_Datatype;
	u64data : LINT;
END_VAR
CASE datatype OF
	OBIS_Datatype.TOTAL_ActiveEnergyPositive:
		u64data := (u64data * 10) / 36;
		u64data := HOST_TO_BE64EX(in := u64data);
		memcpy(srcAddr := ADR(u64data), destAddr := ADR(data[40]), n:= 8);

	OBIS_Datatype.TOTAL_ActiveEnergyNegative:
		u64data := (u64data * 10) / 36;
		u64data := HOST_TO_BE64EX(in := u64data);
		memcpy(srcAddr := ADR(u64data), destAddr := ADR(data[60]), n:= 8);
		
	OBIS_Datatype.TOTAL_ReactiveEnergyPositive:
		u64data := (u64data * 10) / 36;
		u64data := HOST_TO_BE64EX(in := u64data);
		memcpy(srcAddr := ADR(u64data), destAddr := ADR(data[80]), n:= 8);

	OBIS_Datatype.TOTAL_ReactiveEnergyNegative:
		u64data := (u64data * 10) / 36;
		u64data := HOST_TO_BE64EX(in := u64data);
		memcpy(srcAddr := ADR(u64data), destAddr := ADR(data[100]), n:= 8);	

	OBIS_Datatype.TOTAL_ApparentEnergyPositive:
		u64data := (u64data * 10) / 36;
		u64data := HOST_TO_BE64EX(in := u64data);
		memcpy(srcAddr := ADR(u64data), destAddr := ADR(data[120]), n:= 8);

	OBIS_Datatype.TOTAL_ApparentEnergyNegative:
		u64data := (u64data * 10) / 36;
		u64data := HOST_TO_BE64EX(in := u64data);
		memcpy(srcAddr := ADR(u64data), destAddr := ADR(data[140]), n:= 8);		

//--------------------------------------

	OBIS_Datatype.L1_ActiveEnergyPositive:
		u64data := (u64data * 10) / 36;
		u64data := HOST_TO_BE64EX(in := u64data);
		memcpy(srcAddr := ADR(u64data), destAddr := ADR(data[176]), n:= 8);

	OBIS_Datatype.L1_ActiveEnergyNegative:
		u64data := (u64data * 10) / 36;
		u64data := HOST_TO_BE64EX(in := u64data);
		memcpy(srcAddr := ADR(u64data), destAddr := ADR(data[196]), n:= 8);
		
	OBIS_Datatype.L1_ReactiveEnergyPositive:
		u64data := (u64data * 10) / 36;
		u64data := HOST_TO_BE64EX(in := u64data);
		memcpy(srcAddr := ADR(u64data), destAddr := ADR(data[216]), n:= 8);

	OBIS_Datatype.L1_ReactiveEnergyNegative:
		u64data := (u64data * 10) / 36;
		u64data := HOST_TO_BE64EX(in := u64data);
		memcpy(srcAddr := ADR(u64data), destAddr := ADR(data[236]), n:= 8);	

	OBIS_Datatype.L1_ApparentEnergyPositive:
		u64data := (u64data * 10) / 36;
		u64data := HOST_TO_BE64EX(in := u64data);
		memcpy(srcAddr := ADR(u64data), destAddr := ADR(data[256]), n:= 8);

	OBIS_Datatype.L1_ApparentEnergyNegative:
		u64data := (u64data * 10) / 36;
		u64data := HOST_TO_BE64EX(in := u64data);
		memcpy(srcAddr := ADR(u64data), destAddr := ADR(data[276]), n:= 8);		

		
//--------------------------------------

	OBIS_Datatype.L2_ActiveEnergyPositive:
		u64data := (u64data * 10) / 36;
		u64data := HOST_TO_BE64EX(in := u64data);
		memcpy(srcAddr := ADR(u64data), destAddr := ADR(data[320]), n:= 8);

	OBIS_Datatype.L2_ActiveEnergyNegative:
		u64data := (u64data * 10) / 36;
		u64data := HOST_TO_BE64EX(in := u64data);
		memcpy(srcAddr := ADR(u64data), destAddr := ADR(data[340]), n:= 8);
		
	OBIS_Datatype.L2_ReactiveEnergyPositive:
		u64data := (u64data * 10) / 36;
		u64data := HOST_TO_BE64EX(in := u64data);
		memcpy(srcAddr := ADR(u64data), destAddr := ADR(data[360]), n:= 8);

	OBIS_Datatype.L2_ReactiveEnergyNegative:
		u64data := (u64data * 10) / 36;
		u64data := HOST_TO_BE64EX(in := u64data);
		memcpy(srcAddr := ADR(u64data), destAddr := ADR(data[380]), n:= 8);	

	OBIS_Datatype.L2_ApparentEnergyPositive:
		u64data := (u64data * 10) / 36;
		u64data := HOST_TO_BE64EX(in := u64data);
		memcpy(srcAddr := ADR(u64data), destAddr := ADR(data[400]), n:= 8);

	OBIS_Datatype.L2_ApparentEnergyNegative:
		u64data := (u64data * 10) / 36;
		u64data := HOST_TO_BE64EX(in := u64data);
		memcpy(srcAddr := ADR(u64data), destAddr := ADR(data[420]), n:= 8);		

		
		
//--------------------------------------

	OBIS_Datatype.L3_ActiveEnergyPositive:
		u64data := (u64data * 10) / 36;
		u64data := HOST_TO_BE64EX(in := u64data);
		memcpy(srcAddr := ADR(u64data), destAddr := ADR(data[464]), n:= 8);

	OBIS_Datatype.L3_ActiveEnergyNegative:
		u64data := (u64data * 10) / 36;
		u64data := HOST_TO_BE64EX(in := u64data);
		memcpy(srcAddr := ADR(u64data), destAddr := ADR(data[484]), n:= 8);
		
	OBIS_Datatype.L3_ReactiveEnergyPositive:
		u64data := (u64data * 10) / 36;
		u64data := HOST_TO_BE64EX(in := u64data);
		memcpy(srcAddr := ADR(u64data), destAddr := ADR(data[504]), n:= 8);

	OBIS_Datatype.L3_ReactiveEnergyNegative:
		u64data := (u64data * 10) / 36;
		u64data := HOST_TO_BE64EX(in := u64data);
		memcpy(srcAddr := ADR(u64data), destAddr := ADR(data[524]), n:= 8);	

	OBIS_Datatype.L3_ApparentEnergyPositive:
		u64data := (u64data * 10) / 36;
		u64data := HOST_TO_BE64EX(in := u64data);
		memcpy(srcAddr := ADR(u64data), destAddr := ADR(data[544]), n:= 8);

	OBIS_Datatype.L3_ApparentEnergyNegative:
		u64data := (u64data * 10) / 36;
		u64data := HOST_TO_BE64EX(in := u64data);
		memcpy(srcAddr := ADR(u64data), destAddr := ADR(data[564]), n:= 8);			
END_CASE
END_METHOD

METHOD GetData : POINTER TO BYTE
VAR_INPUT
END_VAR
GetData := ADR(data);
END_METHOD

METHOD GetDataLength : UDINT
VAR_INPUT
END_VAR
GetDataLength := 608;
END_METHOD

END_FUNCTION_BLOCK
